VAR_GLOBAL
	
	XTags			: ST_XTags;		

	stVisControl	: ST_VisControl;
	

END_VAR

(* stored: Version 1.1.0.1, ProductVersion 3.1.4024.9
   GVL GlobalVariables: Id {a2a5744c-15c4-44f0-a6cb-58677bd6bb29} *)
